Universal Robots PolyScope program: RC_E3_PICK_320.urp

Program RC_E3_PICK_320 (createdIn=3.0.0 lastSavedIn=3.0.0 directory=/programs installation=default)
Robot Program (runOnlyOnce=true motionType=MoveJ speed=1.047198 acceleration=1.396263 useActiveTCP=false)
  'Program generated by RoboDK v4.1.0 for UR3e_HORNO on 05/09/2022 13:24:50'
  'Using nominal kinematics.'
  'Using Ref. Frame Horno: p[0.203000, 0.332000, 0.148000, 0.000000, 0.000000, 0.000000]'
  'Using TCP 0208-0001-0001-307-000-3 Horno: p[0.000000, 0.000000, 0.164750, 0.000000, 0.000000, 0.000000]'
  Script: set_tcp(p[0.000000, 0.000000, 0.164750, 0.000000, 0.000000, 0.000000])
  Script: movej([1.950645, -1.611670, -0.977770, -2.103192, 1.589544, 0.389279],0.60000,0.12500,0,0.0000)
  Script: movej([1.869632, -2.008207, -0.873961, -1.812100, 1.591139, 0.320999],0.60000,0.12500,0,0.0000)
  MoveL speed 40 mm/s, acceleration 40 mm/s^2 (useActiveTCP=true)
    Waypoint Waypoint_1: TCP in base x=215.764 y=810.562 z=249.954 mm, rx=-3.1288 ry=0.1177 rz=0.0392 rad; joints [103.68, -131.15, -42.93, -94.96, 91.22, 18] deg; flange x=219.825 y=808.71 z=414.644 mm, rx=-3.1288 ry=0.1177 rz=0.0392 rad
  'Attach to 0208-0001-0001-307-000-3 Horno'
  MoveL speed 120 mm/s, acceleration 130 mm/s^2 (useActiveTCP=true)
    Waypoint Waypoint_2: TCP in base x=205.715 y=750.572 z=320.003 mm, rx=-3.1301 ry=0.0344 rz=0.039 rad; joints [107.122, -115.062, -50.074, -103.826, 91.166, 18.392] deg; flange x=209.796 y=748.706 z=484.692 mm, rx=-3.1301 ry=0.0344 rz=0.039 rad
  Script: movej([1.950645, -1.611670, -0.977770, -2.103192, 1.589544, 0.389279],0.13000,0.12000,0,0.0000)
